# EPICS substitutions: apps/jscalerApp/Db/wf/jscalers_wf_S5.substitutions
file "db/jscalers_wf_averages-1type-1sector.db" {
pattern { T S }
{ FADC 5 }
{ TRG 5 }
{ TDC 5 }
}
